(* CODESYS project bl20IoLink.project

Project tree, tasks and I/O mapping:
  Device : BL20-PG-EN-V3, Turck, order no. 6827393, version 3.5.11.20
    application Application
      libraries: Standard, * (System); BLxxFB Local IO, 1.1.1.0 (TURCK)
      task MainTask (cyclic, interval t#20ms, priority 1) calls PLC_PRG
      program PLC_PRG [ST]
    Gateway_LED_APPL : Gateway LED APPL, Turck, version 1.0.3.0
        unmapped channels: Applikation LED (Grün), Applikation LED (Rot), Reserved, Reserved, Reserved, Reserved, Reserved, Reserved
    Local_IO_BL20 : Local IO BL20, Turck, version 1.1.3.0
      BL20_E_4IOL : BL20-E-4IOL, Turck, version 1.1.3.0
          input  Application.PLC_PRG.awLmProcess[0] : WORD  // Input data word 0
          input  Application.PLC_PRG.awLmProcess[1] : WORD  // Input data word 1
          unmapped channels: Input data word 2, Input data word 3, Input data word 4, Input data word 5, Input data word 6, Digital input Ch1, Input value valid Ch1, Digital input Ch2, Input value valid Ch2, Digital input Ch3, Input value valid Ch3, Digital input Ch4, Input value valid Ch4, XSG input Ch5, Overcurrent XSG Ch5, XSG input Ch6, Overcurrent XSG Ch6, XSG input Ch7, Overcurrent XSG Ch7, XSG input Ch8, Overcurrent XSG Ch8, Output data word 0, Output data word 1, Output data word 2, Output data word 3, Output data word 4, Output data word 5, Output data word 6, XSG output Ch5, XSG output Ch6, XSG output Ch7, XSG output Ch8, Dummy, Dummy, Dummy, Dummy, Wrong or missing device Ch1, Data storage error Ch1, Process input data invalid Ch1, Hardware error Ch1,
            Maintenance events Ch1, Out of spec. error Ch1, Parameterization error Ch1, Overtemperature, Lower limit value underrun Ch1, Upper limit value exceeded Ch1, Undervoltage Ch1, Overvoltage Ch1, Overload Ch1, Common error Ch1, Wrong or missing device Ch2, Data storage error Ch2, Process input data invalid Ch2, Hardware error Ch2, Maintenance events Ch2, Out of spec. error Ch2, Parameterization error Ch2, Overtemperature, Lower limit value underrun Ch2, Upper limit value exceeded Ch2, Undervoltage Ch2, Overvoltage Ch2, Overload Ch2, Common error Ch2, Wrong or missing device Ch3, Data storage error Ch3, Process input data invalid Ch3, Hardware error Ch3, Maintenance events Ch3, Out of spec. error Ch3, Parameterization error Ch3, Overtemperature, Lower limit value underrun Ch3, Upper limit value exceeded Ch3, Undervoltage Ch3, Overvoltage Ch3, Overload Ch3, Common error Ch3, Wrong or missing device Ch4, Data storage error Ch4,
            Process input data invalid Ch4, Hardware error Ch4, Maintenance events Ch4, Out of spec. error Ch4, Parameterization error Ch4, Overtemperature, Lower limit value underrun Ch4, Upper limit value exceeded Ch4, Undervoltage Ch4, Overvoltage Ch4, Overload Ch4, Common error Ch4, Overcurrent XSG channel Ch5, Overcurrent XSG channel Ch6, Overcurrent XSG channel Ch7, Overcurrent XSG channel Ch8, Dummy, Dummy, Dummy, Dummy
      BL20_1RS232 : BL20-1RS232, Turck, version 1.1.3.0
          input  Application.PLC_PRG.b232Rx[0] : Byte  // Status byte
          input  Application.PLC_PRG.b232Rx[1] : Byte  // In1 - Diagnostic byte
          input  Application.PLC_PRG.b232Rx[2] : Byte  // In2
          input  Application.PLC_PRG.b232Rx[3] : Byte  // In3
          input  Application.PLC_PRG.b232Rx[4] : Byte  // In4
          input  Application.PLC_PRG.b232Rx[5] : Byte  // In5
          input  Application.PLC_PRG.b232Rx[6] : Byte  // In6
          input  Application.PLC_PRG.b232Rx[7] : Byte  // In7
          output Application.PLC_PRG.b232Tx[0] : Byte  // Control byte
          output Application.PLC_PRG.b232Tx[1] : Byte  // Out1 -ext. control byte
          output Application.PLC_PRG.b232Tx[2] : Byte  // Out2
          output Application.PLC_PRG.b232Tx[3] : Byte  // Out3
          output Application.PLC_PRG.b232Tx[4] : Byte  // Out4
          output Application.PLC_PRG.b232Tx[5] : Byte  // Out5
          output Application.PLC_PRG.b232Tx[6] : Byte  // Out6
          output Application.PLC_PRG.b232Tx[7] : Byte  // Out7
          unmapped channels: Parameterization error, Hardware error, Data flow control error, Frame error, Buffer overflow, Dummy, Dummy, Dummy
    Ethernet : Ethernet, Turck, version 3.5.11.20
      Modbus_TCP_Slave_Device : Modbus TCP Slave Device, Turck, version 1.1.0.0
          output Application.PLC_PRG.awProcessVal[0] : WORD  // Outputs.Outputs
          output Application.PLC_PRG.awProcessVal[1] : WORD  // Outputs.Outputs
          output Application.PLC_PRG.awProcessVal[2] : WORD  // Outputs.Outputs
          output Application.PLC_PRG.awProcessVal[3] : WORD  // Outputs.Outputs
          unmapped channels: Inputs, Outputs
*)

// Device/Application/PLC_PRG
PROGRAM PLC_PRG
VAR CONSTANT
	bCr : BYTE := 13 ;(*CR*)
	bLf : BYTE := 10 ;(*LF*)
	smapleTime : TIME := T#50ms;

END_VAR
VAR
	awLmProcess : ARRAY[0..1] OF WORD; 
	abLmProcess : ARRAY[0..3] OF BYTE;
	rProcessVal : REAL;
	

	rs232Fb : BLxxFB_LIO.BLxx_1RSxxx;
	xEnableRx : BOOL;
	xEnableTx : BOOL := TRUE;
	xQuit : BOOL;
	xClr_Buf_Rx : BOOL;
	xClr_Buf_Tx : BOOL;
	xDisableTxBuffer : BOOL;
	RX_Buffer : ARRAY [0..5] OF BYTE;
	TX_Buffer : ARRAY [0..5] OF BYTE;
	RS232_uiMaxRxByte : UINT := 6;
	RS232_uiMaxTxByte : UINT := 6;
	
	b232Rx : ARRAY[0..7] OF BYTE;
	b232Tx : ARRAY[0..7] OF BYTE;	

	xBusyRx : BOOL;
	xBusyTx : BOOL;
	uiRxBytes :UINT;
	uiTxBytes :UINT;
	xNotEmpty:BOOL;
	wRetVal :WORD;


	tonEnableTx : TON;
	xStart : BOOL;
	tonStart: TON;

	dMeasure : ARRAY[0..2] OF DWORD;
	bMeasure : ARRAY[0..2] OF BYTE;
	wMeasure : ARRAY[0..2] OF WORD;
	dProcessVal : DWORD;
	wProcessVal : WORD;

	bProcessVal : ARRAY[0..3] OF BYTE;
	awProcessVal : ARRAY[0..3] OF WORD;
	
	i : INT;
END_VAR

abLmProcess[0] := WORD_TO_BYTE(awLmProcess[0]/255);
abLmProcess[1] := WORD_TO_BYTE(awLmProcess[0]);
abLmProcess[2] := WORD_TO_BYTE(awLmProcess[1]/255);
abLmProcess[3] := WORD_TO_BYTE(awLmProcess[1]);

bMeasure[0] := SHR(SHL(abLmProcess[1],2),2);
bMeasure[1] := abLmProcess[2];
bMeasure[2] := SHR(abLmProcess[3],3);

FOR i:=0 TO 2 DO
	dMeasure[i] := BYTE_TO_DWORD(bMeasure[i]);
	wMeasure[i] := BYTE_TO_WORD(bMeasure[i]);
END_FOR

dProcessVal := SHL(dMeasure[0],13) + SHL(dMeasure[1], 5) + dMeasure[2];
rProcessVal := DWORD_TO_REAL(dProcessVal)/1000;

bProcessVal[0] := DWORD_TO_BYTE(SHR(dProcessVal, 0));
bProcessVal[1] := DWORD_TO_BYTE(SHR(dProcessVal, 8));
bProcessVal[2] := DWORD_TO_BYTE(SHR(dProcessVal, 16));
bProcessVal[3] := DWORD_TO_BYTE(SHR(dProcessVal, 24));


rs232Fb(xEnableRx := xEnableRx,
		xEnableTx := xEnableTx,
		xQuit := xQuit,
		xClearRxBuffer := xClr_Buf_Rx,
		xClearTxBuffer := xClr_Buf_Tx,
		xDisableTxBuffer := xDisableTxBuffer,
		pbyRxBuffer := ADR(RX_Buffer),
		pbyTxBuffer := ADR(TX_Buffer),
		
		uiMaxRxBytes := RS232_uiMaxRxByte,
		uiMaxTxBytes := RS232_uiMaxTxByte,
		pabyInputData := ADR(b232Rx),
		pabyOutputData := ADR(b232Tx)
);
		
		
xBusyRx := rs232Fb.xBusyRx;
xBusyTx := rs232Fb.xBusyTx;
uiRxBytes := rs232Fb.uiReceivedBytes;
uiTxBytes := rs232Fb.uiSendBytes;
xNotEmpty := rs232Fb.xSendBufNotEmpty;
wRetVal := rs232Fb.wRetVal;

(*
TX_Buffer[0] := bProcessVal[0];
TX_Buffer[1] := bProcessVal[1];
TX_Buffer[2] := bProcessVal[2];
TX_Buffer[3] := bProcessVal[3];
*)
TX_Buffer[4] := bCr;
TX_Buffer[5] := bLf;


tonEnableTx(IN:= xEnableTx, PT := smapleTime);
IF tonEnableTx.Q THEN
	xEnableTx := FALSE;
	xStart := TRUE;
END_IF

tonStart(IN:= xStart, PT := smapleTime);
IF tonStart.Q THEN
	xEnableTx := TRUE;
	xStart := FALSE;
END_IF


FOR i :=0 TO 3 DO
	awProcessVal[i] := bProcessVal[i] ;	
END_FOR

END_PROGRAM
